PROGRAM prgPV
VAR
	fbSE1			: FB_SunSpec_PV_Inverter_T;
	fbSE2			: FB_SunSpec_PV_Inverter_T;
	fbSE3			: FB_SunSpec_PV_Inverter_T;
	fbSE4			: FB_SunSpec_PV_Inverter_T;
	fbPVInt			: FB_PV_Power_Ext_Input;
	fbPVCounter		: FB_EnergyCounter;
	fbPVCounter_1	: FB_EnergyCounter;
	fbPVCounter_2	: FB_EnergyCounter;
	fbPVCounter_3	: FB_EnergyCounter;
	lrPowerPV		: LREAL;					//{#lynus.ag#()}
	lrPowerPV_1		: LREAL;					//{#lynus.ag#()}
	lrPowerPV_2		: LREAL;					//{#lynus.ag#()}
	lrPowerPV_3		: LREAL;					//{#lynus.ag#()}
	lrPowerPV_4		: LREAL;					
	byErrorWarningPV	: BYTE;					//{#lynus.ag#()}
	udintLiveCount		: INT;					//{#lynus.ag#()}
END_VAR
VAR PERSISTENT
	lrCounterPV		: LREAL;					//{#lynus.ag#()}
	lrCounterPV_1	: LREAL;					//{#lynus.ag#()}
	lrCounterPV_2	: LREAL;					//{#lynus.ag#()}
	lrCounterPV_3	: LREAL;					//{#lynus.ag#()}
END_VAR

fbSE1(
	bEnable:= TRUE, 
	sIPAdress:= '192.168.44.45', 
	byUnitID_Inverter:= 1, 
	stDataSunSpec=> , 
	stDataEMPower_PV=> , 
	stDataEMCounter_PV=> , 
	diNrOfEM_OUT_PV=> );
	
fbSE2(
	bEnable:= TRUE, 
	sIPAdress:= '192.168.44.46', 
	byUnitID_Inverter:= 1, 
	stDataSunSpec=> , 
	stDataEMPower_PV=> , 
	stDataEMCounter_PV=> , 
	diNrOfEM_OUT_PV=> );
	
fbSE3(
	bEnable:= TRUE, 
	sIPAdress:= '192.168.44.50', 
	byUnitID_Inverter:= 1, 
	stDataSunSpec=> , 
	stDataEMPower_PV=> , 
	stDataEMCounter_PV=> , 
	diNrOfEM_OUT_PV=> );

fbSE4(
	bEnable:= FALSE, 
	sIPAdress:= '192.168.44.50', 
	byUnitID_Inverter:= 2, 
	stDataSunSpec=> , 
	stDataEMPower_PV=> , 
	stDataEMCounter_PV=> , 
	diNrOfEM_OUT_PV=> );
	
lrPowerPV_1 := fbSE1.stDataEMPower_PV.lrPowerTotal;
lrPowerPV_2 := fbSE2.stDataEMPower_PV.lrPowerTotal;
lrPowerPV_3 := fbSE3.stDataEMPower_PV.lrPowerTotal;
lrPowerPV_4 := fbSE4.stDataEMPower_PV.lrPowerTotal;
lrCounterPV_1 := fbSE1.stDataEMCounter_PV.lrCounterEnergyT1_Production;
lrCounterPV_2 := fbSE2.stDataEMCounter_PV.lrCounterEnergyT1_Production;
lrCounterPV_3 := fbSE3.stDataEMCounter_PV.lrCounterEnergyT1_Production;
	
fbPVInt(
	bEnable:= TRUE, 
	bExtErrorPV := , 
	lrExtPvPower := lrPowerPV_1 + lrPowerPV_2 + lrPowerPV_3, 
	stDataPv=> , 
	diNrOfPv_OUT=> );
	
lrPowerPV := fbPVInt.stDataPv.lrPower;
	byErrorWarningPV := fbPVInt.stDataPv.byErrorWarning;
	

// for testing purpose

udintLiveCount := udintLiveCount+1;

END_PROGRAM

(* stored: Version 1.1.0.1, ProductVersion 3.1.4024.12
   POU prgPV: Id {52a4cf08-62d2-4b94-900b-2ea0759cae15}, SpecialFunc None *)
